// Mitsubishi GX Works2 project: 译码顺控   PLC: FX3G

PROGRAM MAIN
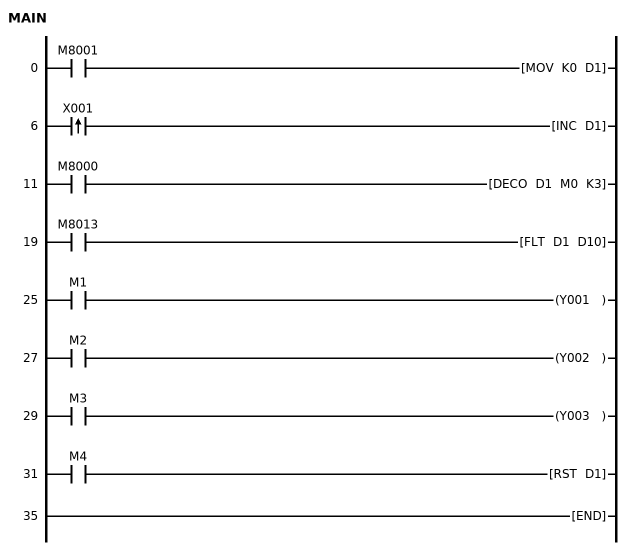
0     LD      M8001
      MOV     K0 D1
6     LDP     X001
      INC     D1
11    LD      M8000
      DECO    D1 M0 K3
19    LD      M8013
      FLT     D1 D10
25    LD      M1
      OUT     Y001
27    LD      M2
      OUT     Y002
29    LD      M3
      OUT     Y003
31    LD      M4
      RST     D1
35    END
END_PROGRAM
